(* PLC project Blink_Pox_2017_02, FGDES/LRT CompileDES 3.10 *)
(* stored: creationDateTime 2017-03-14T15:42:55 *)

FUNCTION_BLOCK fcg_cyclic_fb
  VAR_INPUT
    RESET : BOOL := false;  (* external reset *)
  END_VAR
  VAR_OUTPUT
    STATUS : BYTE;  (* status (0x00 <> waiting, 0x01<>executing, 0x02<>err) *)
    RECENT_EVENT : INT;  (* recent event (0<>none) *)
    PENDING_EVENTS : ARRAY[0..0] OF BYTE;  (* pending input events incl timer elapse *)
    ENABLED_EVENTS : ARRAY[0..0] OF BYTE;  (* events enabled by all generators *)
    PARALLEL_STATE : ARRAY[0..2] OF INT;  (* parallel state *)
  END_VAR
  VAR
    fcg_exec_event : INT := -1;  (* executed event (-1<>init, 0<>none) *)
    fcg_sched_event : INT;  (* scheduled event (0<>none) *)
    fcg_line_level_0 : BOOL;  (* line levels *)
    fcg_first_loop : BOOL;  (* loop flag *)
    fcg_timer_Tick_cnt : TIME;  (* timer states *)
    fcg_timer_Tick_run : BOOL;  (* timer states *)
    fcg_time_elapsed : TIME;  (* elapsed time since last invokation *)
    fcg_aux_locenabled : ARRAY[0..0] OF BYTE;  (* parse generator *)
    fcg_aux_parsetrans : INT;  (* parse generator *)
    fcg_aux_parseevent : INT;  (* parse generator *)
    fcg_aux_executables : ARRAY[0..0] OF BYTE;  (* enabled events that can be executed *)
    fcg_aux_wordret : BYTE;  (* aux maths and stack variables *)
    fcg_aux_edge : BOOL;  (* aux maths and stack variables *)
    fcg_aux_wordaddr : INT;  (* aux maths and stack variables *)
    fcg_aux_bitaddr : INT;  (* aux maths and stack variables *)
    fcg_aux_bitmask : BYTE;  (* aux maths and stack variables *)
    fcg_bitmask_vector : ARRAY[0..7] OF BYTE := [BYTE#16#01, BYTE#16#02, BYTE#16#04, BYTE#16#08, BYTE#16#10, BYTE#16#20, BYTE#16#40, BYTE#16#80];  (* mask vectors *)
    fcg_generator_states_0 : ARRAY[1..6] OF INT := [0, 3, 6, 9, 12, 15];  (* generator [Blink3] *)
    fcg_generator_transitions_0 : ARRAY[0..17] OF INT := [3, 2, 0, 4, 3, 0, 5, 6, 0, 7, 5, 0, 8, 1, 0, 6, 4, 0];  (* generator [Blink3] *)
    fcg_generator_transitions_1 : ARRAY[0..15] OF INT := [3, 13, 4, 13, 5, 13, 6, 13, 7, 13, 8, 13, 0, 2, 0, 0];  (* generator [Delay] *)
    fcg_generator_transitions_2 : ARRAY[0..11] OF INT := [6, 0, 1, 5, 0, 3, 5, 6, 0, 1, 5, 0];  (* generator [WaitButton] *)
    fcg_systime_ton : TON;  (* iec timer to simulate system time *)
    fcg_systime_recent : TIME;  (* iec timer to simulate system time *)
    fcg_systime_now : TIME;  (* iec timer to simulate system time *)
  END_VAR
  VAR_EXTERNAL
    input : BOOL;  (* import i/o variables and addresses *)
  END_VAR

(* ************************************************ *)
(* CodeGenerator: Target IEC 61131 Structured Text  *)
(* ************************************************ *)


(* CompileDES 3.10 (using libFAUDES 2.28a) *)
(* Configuration: Blink_Pox_2017_02 *)



(* ************************************************ *)
(* * executor core cyclic code: reset/initialise  * *)
(* ************************************************ *)


(* ************************************************ *)
(* * reset internal state                         * *)

(* set internal reset flag *)
IF RESET THEN
    fcg_exec_event := -1;
END_IF;

(* do reset core *)
IF fcg_exec_event = -1 THEN
  (* clear status *)
  STATUS := 0;
  (* set initial state *)
  PARALLEL_STATE[0] := 1;
  PARALLEL_STATE[1] := 0;
  PARALLEL_STATE[2] := 0;
  (* clear scheduled event *)
  fcg_sched_event := 0;
  (* clear recent event *)
  RECENT_EVENT := 0;
  (* clear pending/enabled events *)
  PENDING_EVENTS[0] := BYTE#0;
  ENABLED_EVENTS[0] := BYTE#0;
  (* reset timer *)
  fcg_timer_Tick_run := false;
  fcg_timer_Tick_cnt := TIME#1s;
END_IF;

(* do reset/track systime *)
IF fcg_exec_event = -1  THEN
  fcg_systime_ton(IN:=false);
  fcg_systime_recent := TIME#0ms;
END_IF;
fcg_systime_ton(IN:=true, PT:=TIME#2h, ET=>fcg_systime_now);
fcg_time_elapsed := fcg_systime_now - fcg_systime_recent;
IF fcg_systime_now < TIME#1h THEN
  fcg_systime_recent := fcg_systime_now;
ELSE
  fcg_systime_ton(IN:=false, PT:=TIME#2h);
  fcg_systime_ton(IN:=true, PT:=TIME#2h);
  fcg_systime_recent := TIME#0ms;
END_IF;



(* ************************************************ *)
(* * bail out on external reset                   * *)

IF RESET THEN
    RETURN;
END_IF;



(* ************************************************ *)
(* * update timer states                          * *)


IF fcg_time_elapsed > TIME#0ms THEN
  IF fcg_timer_Tick_run THEN
    IF fcg_timer_Tick_cnt > fcg_time_elapsed THEN
      fcg_timer_Tick_cnt := fcg_timer_Tick_cnt - fcg_time_elapsed;
    ELSE
      fcg_timer_Tick_cnt := TIME#0s;
    END_IF;
  END_IF;
END_IF;



(* ************************************************ *)
(* * executor core cyclic code: begin             * *)
(* ************************************************ *)



(* ************************************************ *)
(* * sense input events                           * *)

(* init: reset all line data and generate statics *)
IF fcg_exec_event = -1 THEN
  fcg_line_level_0 := input;
  IF fcg_line_level_0 THEN
    (* positive value: trigger init event [PushButton] *)
    PENDING_EVENTS[0] := PENDING_EVENTS[0] OR BYTE#16#01;
  END_IF;
END_IF;

(* normal operation: read lines and detect edges *)
IF fcg_exec_event <> -1 THEN
  (* read line [input] *)
  fcg_aux_edge := input;
  IF fcg_aux_edge <> fcg_line_level_0 THEN
    IF fcg_aux_edge THEN
      (* positive edge: trigger input event [PushButton] *)
      PENDING_EVENTS[0] := PENDING_EVENTS[0] OR BYTE#16#01;
      fcg_sched_event := 0;
    END_IF;
    fcg_line_level_0 := fcg_aux_edge;
  END_IF;
END_IF;



(* ************************************************ *)
(* * sense timer elapse                           * *)

IF fcg_timer_Tick_run AND (fcg_timer_Tick_cnt <= TIME#0ms) THEN
  fcg_timer_Tick_run := false;
  PENDING_EVENTS[0] := PENDING_EVENTS[0] OR BYTE#16#02;
  fcg_sched_event := 0;
END_IF;



(* ************************************************ *)
(* * event execution loop                         * *)

(* clear status to waiting *)
STATUS := 0;
(* clear event report *)
RECENT_EVENT := 0;
(* set entry flag *)
fcg_first_loop := true;
WHILE true DO



(* ************************************************ *)
(* * update enabled events after execution        * *)

(* if event was executed (and on init) *)
IF fcg_exec_event <> 0 THEN

  (* set all to enabled *)
  ENABLED_EVENTS[0] := BYTE#16#ff;

  (* setup enabled events by [Blink3] *)
  fcg_aux_locenabled[0] := BYTE#16#03;
  fcg_aux_parsetrans := fcg_generator_states_0[PARALLEL_STATE[0]];
  WHILE true DO
    fcg_aux_parseevent := fcg_generator_transitions_0[fcg_aux_parsetrans];
    IF fcg_aux_parseevent = 0 THEN EXIT; END_IF;
    fcg_aux_bitaddr := fcg_aux_parseevent;
    fcg_aux_bitaddr := fcg_aux_bitaddr - 1;
    fcg_aux_bitmask := fcg_bitmask_vector[fcg_aux_bitaddr];
    fcg_aux_locenabled[fcg_aux_wordaddr] := fcg_aux_locenabled[fcg_aux_wordaddr] OR fcg_aux_bitmask;
    fcg_aux_parsetrans := fcg_aux_parsetrans + 2;
  END_WHILE;
  (* restrict enabled events *)
  ENABLED_EVENTS[0] := ENABLED_EVENTS[0] AND fcg_aux_locenabled[0];

  (* setup enabled events by [Delay] *)
  fcg_aux_locenabled[0] := BYTE#16#01;
  fcg_aux_parsetrans := PARALLEL_STATE[1];
  WHILE true DO
    fcg_aux_parseevent := fcg_generator_transitions_1[fcg_aux_parsetrans];
    IF fcg_aux_parseevent = 0 THEN EXIT; END_IF;
    fcg_aux_bitaddr := fcg_aux_parseevent;
    fcg_aux_bitaddr := fcg_aux_bitaddr - 1;
    fcg_aux_bitmask := fcg_bitmask_vector[fcg_aux_bitaddr];
    fcg_aux_locenabled[fcg_aux_wordaddr] := fcg_aux_locenabled[fcg_aux_wordaddr] OR fcg_aux_bitmask;
    fcg_aux_parsetrans := fcg_aux_parsetrans + 2;
  END_WHILE;
  (* restrict enabled events *)
  ENABLED_EVENTS[0] := ENABLED_EVENTS[0] AND fcg_aux_locenabled[0];

  (* setup enabled events by [WaitButton] *)
  fcg_aux_locenabled[0] := BYTE#16#da;
  fcg_aux_parsetrans := PARALLEL_STATE[2];
  WHILE true DO
    fcg_aux_parseevent := fcg_generator_transitions_2[fcg_aux_parsetrans];
    IF fcg_aux_parseevent = 0 THEN EXIT; END_IF;
    fcg_aux_bitaddr := fcg_aux_parseevent;
    fcg_aux_bitaddr := fcg_aux_bitaddr - 1;
    fcg_aux_bitmask := fcg_bitmask_vector[fcg_aux_bitaddr];
    fcg_aux_locenabled[fcg_aux_wordaddr] := fcg_aux_locenabled[fcg_aux_wordaddr] OR fcg_aux_bitmask;
    fcg_aux_parsetrans := fcg_aux_parsetrans + 2;
  END_WHILE;
  (* restrict enabled events *)
  ENABLED_EVENTS[0] := ENABLED_EVENTS[0] AND fcg_aux_locenabled[0];

  (* dispose event *)
  fcg_exec_event := 0;
  fcg_sched_event := 0;
END_IF;



(* ************************************************ *)
(* * schedule next event to execute               * *)

IF fcg_sched_event = 0 THEN

  (* setup candidate set to "pending or internal" *)
  fcg_aux_executables[0] := PENDING_EVENTS[0] OR BYTE#16#fc;
  (* restrict candidate set by "enabled" *)
  fcg_aux_executables[0] := fcg_aux_executables[0] AND ENABLED_EVENTS[0];

  (* find highest priority event (lowest bitaddress) *)
  fcg_sched_event := 0;
  IF NOT ( fcg_aux_executables[0] = BYTE#0 ) THEN
    IF ( fcg_aux_executables[0] AND BYTE#16#0f ) <> BYTE#0 THEN
      IF ( fcg_aux_executables[0] AND BYTE#16#03 ) <> BYTE#0 THEN
        IF ( fcg_aux_executables[0] AND BYTE#16#01 ) <> BYTE#0 THEN
          fcg_sched_event := 1;
        ELSE
          fcg_sched_event := 2;
        END_IF;
      ELSE
        IF ( fcg_aux_executables[0] AND BYTE#16#04 ) <> BYTE#0 THEN
          fcg_sched_event := 3;
        ELSE
          fcg_sched_event := 4;
        END_IF;
      END_IF;
    ELSE
      IF ( fcg_aux_executables[0] AND BYTE#16#30 ) <> BYTE#0 THEN
        IF ( fcg_aux_executables[0] AND BYTE#16#10 ) <> BYTE#0 THEN
          fcg_sched_event := 5;
        ELSE
          fcg_sched_event := 6;
        END_IF;
      ELSE
        IF ( fcg_aux_executables[0] AND BYTE#16#40 ) <> BYTE#0 THEN
          fcg_sched_event := 7;
        ELSE
          fcg_sched_event := 8;
        END_IF;
      END_IF;
    END_IF;
  END_IF;

  (* remove scheduled event from pending events *)
  IF fcg_sched_event > 0 THEN
    fcg_aux_bitaddr := fcg_sched_event;
    fcg_aux_bitaddr := fcg_aux_bitaddr - 1;
    fcg_aux_bitmask := fcg_bitmask_vector[fcg_aux_bitaddr];
    PENDING_EVENTS[fcg_aux_wordaddr] := PENDING_EVENTS[fcg_aux_wordaddr] AND (NOT fcg_aux_bitmask );
  END_IF;

  (* detect sync error *)
  IF fcg_sched_event = 0 THEN
    fcg_aux_wordret := PENDING_EVENTS[0];
    IF NOT ( fcg_aux_wordret = BYTE#0 ) THEN
      STATUS := STATUS OR BYTE#16#02;
    END_IF;
  END_IF;

  (* cancel pending events if no event could be scheduled  *)
  IF fcg_sched_event = 0 THEN
    PENDING_EVENTS[0] := BYTE#0;
  END_IF;

END_IF;



(* ************************************************ *)
(* * break execution loop                         * *)

IF fcg_sched_event = 0 THEN EXIT; END_IF;
fcg_first_loop := false;



(* ************************************************ *)
(* * execute scheduled event                      * *)

IF fcg_sched_event <> 0 THEN

  fcg_exec_event := fcg_sched_event;
  fcg_sched_event := 0;
  STATUS := STATUS OR BYTE#16#01;

  (* execute event for [Blink3] *)
  fcg_aux_parsetrans := fcg_generator_states_0[PARALLEL_STATE[0]];
  WHILE true DO
    fcg_aux_parseevent := fcg_generator_transitions_0[fcg_aux_parsetrans];
    IF fcg_aux_parseevent = fcg_exec_event THEN EXIT; END_IF;
    IF fcg_aux_parseevent = 0 THEN EXIT; END_IF;
    fcg_aux_parsetrans := fcg_aux_parsetrans + 2;
  END_WHILE;
  IF fcg_aux_parseevent > 0 THEN
    fcg_aux_parsetrans := fcg_aux_parsetrans + 1;
    PARALLEL_STATE[0] := fcg_generator_transitions_0[fcg_aux_parsetrans];
  END_IF;

  (* execute event for [Delay] *)
  fcg_aux_parsetrans := PARALLEL_STATE[1];
  WHILE true DO
    fcg_aux_parseevent := fcg_generator_transitions_1[fcg_aux_parsetrans];
    IF fcg_aux_parseevent = fcg_exec_event THEN EXIT; END_IF;
    IF fcg_aux_parseevent = 0 THEN EXIT; END_IF;
    fcg_aux_parsetrans := fcg_aux_parsetrans + 2;
  END_WHILE;
  IF fcg_aux_parseevent > 0 THEN
    fcg_aux_parsetrans := fcg_aux_parsetrans + 1;
    PARALLEL_STATE[1] := fcg_generator_transitions_1[fcg_aux_parsetrans];
  END_IF;

  (* execute event for [WaitButton] *)
  fcg_aux_parsetrans := PARALLEL_STATE[2];
  WHILE true DO
    fcg_aux_parseevent := fcg_generator_transitions_2[fcg_aux_parsetrans];
    IF fcg_aux_parseevent = fcg_exec_event THEN EXIT; END_IF;
    IF fcg_aux_parseevent = 0 THEN EXIT; END_IF;
    fcg_aux_parsetrans := fcg_aux_parsetrans + 2;
  END_WHILE;
  IF fcg_aux_parseevent > 0 THEN
    fcg_aux_parsetrans := fcg_aux_parsetrans + 1;
    PARALLEL_STATE[2] := fcg_generator_transitions_2[fcg_aux_parsetrans];
  END_IF;

  (* record *)
  RECENT_EVENT := fcg_exec_event;

END_IF;



(* ************************************************ *)
(* * operate timers                               * *)

IF fcg_exec_event > 0 THEN
  CASE fcg_exec_event OF
  3 .. 8:
    fcg_timer_Tick_cnt := TIME#1s;
    fcg_timer_Tick_run := true;
  END_CASE;
END_IF;



(* ************************************************ *)
(* * operate outputs                              * *)

IF fcg_exec_event > 2 THEN
  CASE fcg_exec_event OF
  3:
    (* outputs for [OnLedA] *)
    %QX55.1 := true;
  4:
    (* outputs for [OnLedB] *)
    %QX55.2 := true;
  5:
    (* outputs for [OnLedC] *)
    %QX55.3 := true;
  6:
    (* outputs for [OffLedA] *)
    %QX55.1 := false;
  7:
    (* outputs for [OffLedB] *)
    %QX55.2 := false;
  8:
    (* outputs for [OffLedC] *)
    %QX55.3 := false;
  END_CASE;
END_IF;



(* ************************************************ *)
(* * end execution loop                           * *)

END_WHILE;




(* ************************************************ *)
(* * executor core cyclic code: end               * *)
(* ************************************************ *)



(* ************************************************ *)
(* CodeGenerator: Generated Code Ends Here          *)
(* ************************************************ *)
END_FUNCTION_BLOCK

FUNCTION fcg_event_lookup_f : STRING
  VAR_INPUT
    IDX : INT;  (* event index *)
  END_VAR
  VAR CONSTANT
    fcg_event_lookup : ARRAY[1..8] OF STRING(10) := ['PushButton', 'Tick', 'OnLedA', 'OnLedB', 'OnLedC', 'OffLedA', 'OffLedB', 'OffLedC'];  (* event name lookup table *)
  END_VAR

fcg_event_lookup_f := fcg_event_lookup[IDX];
END_FUNCTION

FUNCTION fcg_state_lookup_f : STRING
  VAR_INPUT
    GID : INT;  (* generator id *)
    IDX : INT;  (* state index *)
  END_VAR
  VAR CONSTANT
    fcg_state_lookup_0 : ARRAY[1..6] OF STRING(4) := ['On0', 'On1', 'On2', 'Off2', 'Off1', '#6'];  (* state name lookup for generator [Blink3] *)
  END_VAR

fcg_state_lookup_f:='';
CASE GID OF
0: fcg_state_lookup_f := fcg_state_lookup_0[IDX];


END_CASE;
IF LEN(fcg_state_lookup_f) = 0 THEN
  fcg_state_lookup_f := CONCAT('s',INT_TO_STRING(IDX));
END_IF;
END_FUNCTION
